FUNCTION_BLOCK GreenWhiteBackgroundAux (* Composite FB wrapping other FBs *)
  (* Standard: 61499-2 *)
  (* Version 1.0, 2022-11-10, franz *)
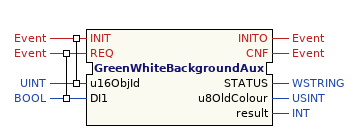
  EVENT_INPUT
    INIT WITH u16ObjId; (* Initialization Request *)
    REQ WITH DI1; (* Normal Execution Request *)
  END_EVENT
  EVENT_OUTPUT
    INITO; (* Initialization Confirm *)
    CNF; (* Execution Confirmation *)
  END_EVENT
  VAR_INPUT
    u16ObjId : UINT; (* Object ID *)
    DI1 : BOOL; (* Selelctor *)
  END_VAR
  VAR_OUTPUT
    STATUS : WSTRING; (* Service Status *)
    u8OldColour : USINT; (* Old value of ID *)
    result : INT; (* retval see description *)
  END_VAR
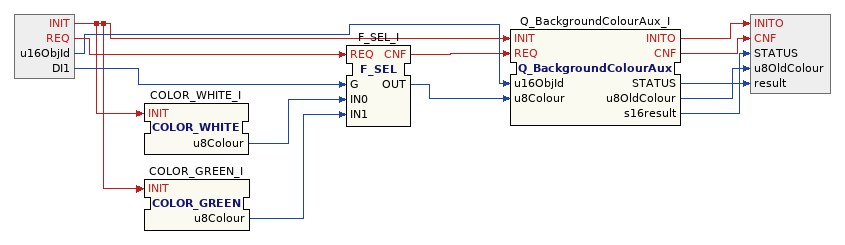
  FBS
    F_SEL_I : F_SEL;
    COLOR_WHITE_I : COLOR_WHITE;
    COLOR_GREEN_I : COLOR_GREEN;
    Q_BackgroundColourAux_I : Q_BackgroundColourAux;
  END_FBS
  EVENT_CONNECTIONS
    REQ TO F_SEL_I.REQ;
    INIT TO COLOR_WHITE_I.INIT;
    INIT TO COLOR_GREEN_I.INIT;
    INIT TO Q_BackgroundColourAux_I.INIT;
    F_SEL_I.CNF TO Q_BackgroundColourAux_I.REQ;
    Q_BackgroundColourAux_I.INITO TO INITO;
    Q_BackgroundColourAux_I.CNF TO CNF;
  END_CONNECTIONS
  DATA_CONNECTIONS
    DI1 TO F_SEL_I.G;
    COLOR_WHITE_I.u8Colour TO F_SEL_I.IN0;
    COLOR_GREEN_I.u8Colour TO F_SEL_I.IN1;
    u16ObjId TO Q_BackgroundColourAux_I.u16ObjId;
    F_SEL_I.OUT TO Q_BackgroundColourAux_I.u8Colour;
    Q_BackgroundColourAux_I.STATUS TO STATUS;
    Q_BackgroundColourAux_I.u8OldColour TO u8OldColour;
    Q_BackgroundColourAux_I.s16result TO result;
  END_CONNECTIONS
END_FUNCTION_BLOCK
